// TIA Portal V19 export
TYPE "LAF_typePlcDiag"
TITLE = PLC Diag
// Type contains all information of the PLC diagnostic which will be displayed at the HMI. / PLC Informationen fuer HMI
// stored: Access Published
   STRUCT
      manualReadAll : Bool;   // Manueller Anstoss; erneutes Einlesen aller Daten/Infos / Manual trigger; renew informations
      blockBusyAfterRestart : Bool;   // FB_Busy nach Neustart / FB busy after restart
      im0Data : IM0_Data;   // I&M 0-Daten / I&M 0-Data
      im1PlantDesignLocIdent : String[54];   // I&M 1-Daten: Anlagen- und Ortskennzeichen / I&M 1-Data: Plant designation & Location identifier
      im1PlantDesignation : String[54];   // I&M 1-Daten: Anlagenkennzeichen / I&M 1-Data: Plant designation
      im1LocIdent : String[54];   // I&M 1-Daten: Ortskennzeichen / I&M 1-Data: Location identifier
      im2InstallationDate : String[54];   // I&M 2-Daten / I&M 2-Data: Installation date
      im3AdditionalInfo : String[54];   // I&M 3-Daten / I&M 3-Data: Additional Info
      addressMac : Array[0..5] of Byte;   // MAC/Ethernet-Adresse / MAC/Ethernet address
      addressIpV4 : Array[0..3] of USInt;   // IPv4-Adresse / IP v4 address
      addressSubnet : Array[0..3] of USInt;   // Subnet-Adresse / Subnet-address
      im0SwRev : String[1];   // für Visualisierung (Wandlung auf String) / For visualization
   END_STRUCT;
END_TYPE
